// Structured view.
FUNCTION_BLOCK FB_Mfr_View EXTENDS FB_Mfr

SUPER^();

END_FUNCTION_BLOCK

(* stored: Version 1.1.0.1
   POU FB_Mfr_View: Id {1e8dc142-ac54-4a17-a957-efb30e95be83}, SpecialFunc None *)
